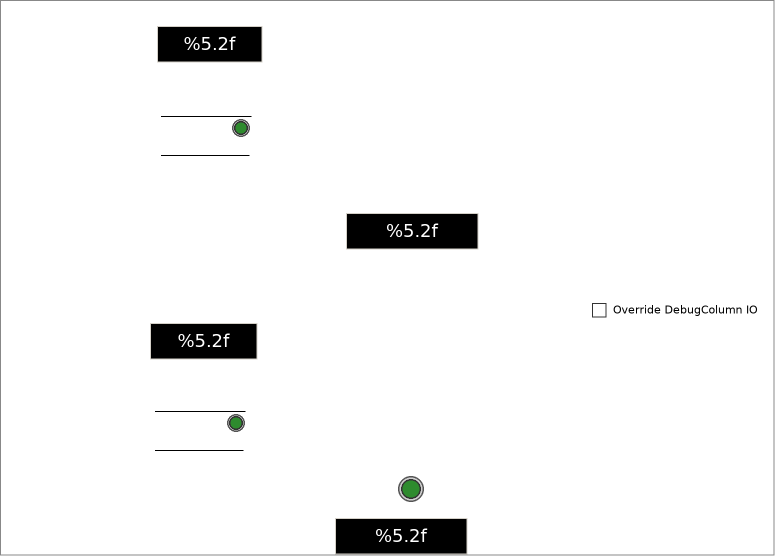
VISUALIZATION HMI_OFA_Monitor  // 775x556, background image ImageCollection.OFA Flow
    Lamp1 (396,474 30x30), variable: stDebugStation.fbDBStnSeq.stDebugStationDIO.opDBStnBypassAPAirSupplySol, style: Lamp-Lamp1-Green
    Textfield (157,26 105x36), "%5.2f", text variable: fbDebugColumn.stDebugColumnDIO.ipDBColumnTstAirPressure, input disabled if: TRUE
    Textfield (150,323 107x36), "%5.2f", text variable: fbDebugColumn.stDebugColumnDIO.ipDBColumnAPAirPressure, input disabled if: TRUE
    Rectangle (296,39 439x145)
    Rectangle (289,335 439x120)
    Lamp1 (226,413 20x20), variable: fbDebugColumn.stDebugColumnDIO.opDBColumnAPAirSol, style: Lamp-Lamp1-Green
    Lamp1 (231,118 20x20), variable: fbDebugColumn.stDebugColumnDIO.opDBColumnTstAirSol, style: Lamp-Lamp1-Green
    Textfield (346,213 132x36), "%5.2f", text variable: stDebugStation.fbDBStnSeq.stDebugStationDIO.ipDBStnTstAirLeakFlowSensor, input disabled if: TRUE
    Textfield (335,518 132x36), "%5.2f", text variable: stDebugStation.fbDBStnSeq.stDebugStationDIO.ipDBStnAPAirLeakFlowSensor, input disabled if: TRUE
    Line (155,411) (245,411)
    Line (155,450) (243,450)
    Line (161,116) (251,116)
    Line (161,155) (249,155)
    Checkbox (590,295 183x30), "Override DebugColumn IO"
END_VISUALIZATION

(* stored: Version 1.1.0.1, ProductVersion 3.1.4022.12
   Visu HMI_OFA_Monitor: Id {16615568-e8eb-4733-a79b-6d37bda70eaa} *)
